FUNCTION_BLOCK AB_TO_AB2 (* Composite FB for convert unidirectional AB to bidirectional AB2 *)
  (* Standard: 61499-2; Function: AB_IN publishes its value onto the outgoing (EO1) side of AB2_BIDIR. Whatever AB2_BIDIR receives on its incoming (EI1) side is forwarded out again as a plain unidirectional signal via AB_OUT.; Description: Copyright (c) 2026 HR Agrartechnik GmbH This program and the accompanying materials are made available under the terms of the Eclipse Public License 2.0 which is available at https://www.eclipse.org/legal/epl-2.0/ SPDX-License-Identifier: EPL-2.0 *)
  (* Version 1.0, 2026-08-31, Franz Höpfinger, HR Agrartechnik GmbH, Initial Version *)
  PACKAGE adapter::conversion::bidirectional;
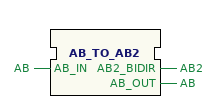
  SOCKETS
    AB_IN : adapter::types::unidirectional::AB; (* Adapter Input: unidirectional source *)
  END_SOCKETS
  PLUGS
    AB2_BIDIR : adapter::types::bidirectional::AB2; (* Adapter Output: bidirectional tap, outgoing side driven by AB_IN, incoming side forwarded to AB_OUT *)
    AB_OUT : adapter::types::unidirectional::AB; (* Adapter Output: mirrors AB2_BIDIR's incoming (request) side *)
  END_PLUGS
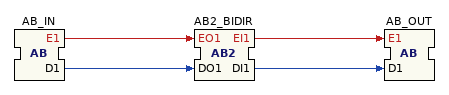
  EVENT_CONNECTIONS
    AB_IN.E1 TO AB2_BIDIR.EO1;
    AB2_BIDIR.EI1 TO AB_OUT.E1;
  END_CONNECTIONS
  DATA_CONNECTIONS
    AB_IN.D1 TO AB2_BIDIR.DO1;
    AB2_BIDIR.DI1 TO AB_OUT.D1;
  END_CONNECTIONS
END_FUNCTION_BLOCK
